Yaskawa INFORM job: test1.jbi

/JOB
//NAME test1
//POS
///NPOS 0,0,0,0,0,0
//INST
///DATE 2021/01/13 23:21
///ATTR SC,RW
///LVARS 3,3,3,3,0,0,0,0
NOP
MOVJ P012 VJ=123.00 //jfdkdsjfk
MOVL P0123  V=120.0 //dsdsdsa



SET B012  EXPRESS B012 + B012 + (LI001) * 1000
SET Bxxx  EXPRESS expression
SET LD123 B123
SETULAM 8123 "dfdsfds" 1
WAIT IN#(1) T=12.00
MOVJ P012 BP012 VJ=12.00 //fgfdgdf
MOVJ P012 VJ=12.00 //dsgdsfffds
GETS LPX012 $PX011
GETE LD000 P012 (1)
GETE LD001 P012 (2)
GETE LD002 P012 (3)
SETE LD000  EXPRESS LD000 + ( 12 ) * 1000
SETE LD001  EXPRESS LD001 + ( 13 ) * 1000
SETE LD002  EXPRESS LD002 + ( 134 ) * 1000
SETE P012 (1) LD000
SETE P012 (2) LD001
SETE P012 (3) LD002
FOR LI000 START= 12 TO 90 STEP=2
    SET P0[LI000] P0[L]

NEXT LI000

SWITCH LI000
CASE <value>

DEFAULT
ENDSWITCH





END
